{attribute 'qualified_only'}
VAR_GLOBAL CONSTANT
	MAX_TANK		: UDINT := 3;
END_VAR

(* stored: Version 1.1.0.1
   GVL CST: Id {6f97e508-fbf2-4606-b6a8-4e1cef309f6b} *)
